Omron CX-Programmer project NewProject (CX-Programmer 9.61)

# PLC AX10: CP1H XA

## Global symbols (name address type ; comment)
0.00 BOOL  ; SENS_1
0.01 BOOL  ; DETECT
0.02 BOOL  ; SENS_2
0.03 BOOL  ; Z_MOV
0.04 BOOL  ; X_MOV
0.05 BOOL  ; START_BT
100.00 BOOL  ; CON
100.01 BOOL  ; Z_AXIS
100.02 BOOL  ; GRAB
100.03 BOOL  ; X_AXIS
100.04 BOOL  ; ROLL
100.05 BOOL  ; CONV_2
100.06 BOOL  ; CONV_3
10.00 BOOL  ; O1
10.01 BOOL  ; O2
10.02 BOOL  ; O3
10.03 BOOL  ; O4
10.04 BOOL  ; O5
T0000 BOOL  ; TIM_1
T0001 BOOL  ; TIM_2
T0002 BOOL  ; TIM_3
T0003 BOOL  ; TIM_4
T0004 BOOL  ; TIM_5
T0005 BOOL  ; TIM_6
T0006 BOOL  ; TIM_7
T0008 BOOL  ; TIM_8
T0009 BOOL  ; TIM_9

## Program NewProgram1 (cyclic task 0)
Local symbols
TOO6 BOOL

### Section Section1

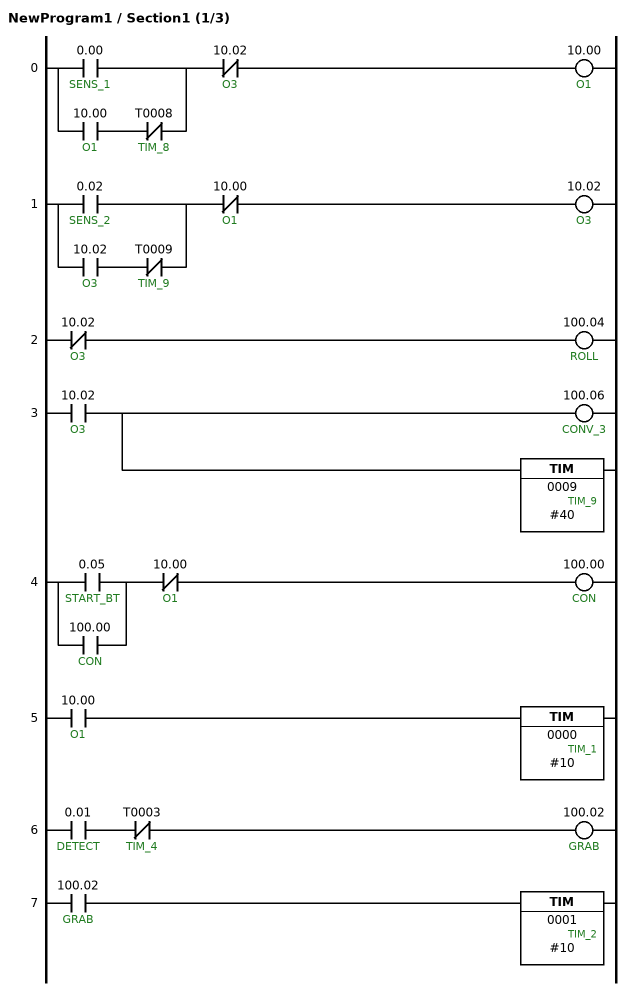
; rung 0
LD 0.00  ; SENS_1
LD 10.00  ; O1
ANDNOT T0008  ; TIM_8
ORLD
ANDNOT 10.02  ; O3
OUT 10.00  ; O1
; rung 1
LD 0.02  ; SENS_2
LD 10.02  ; O3
ANDNOT T0009  ; TIM_9
ORLD
ANDNOT 10.00  ; O1
OUT 10.02  ; O3
; rung 2
LDNOT 10.02  ; O3
OUT 100.04  ; ROLL
; rung 3
LD 10.02  ; O3
OUT 100.06  ; CONV_3
TIM 0009 #40  ; TIM_9
; rung 4
LD 0.05  ; START_BT
OR 100.00  ; CON
ANDNOT 10.00  ; O1
OUT 100.00  ; CON
; rung 5
LD 10.00  ; O1
TIM 0000 #10  ; TIM_1
; rung 6
LD 0.01  ; DETECT
ANDNOT T0003  ; TIM_4
OUT 100.02  ; GRAB
; rung 7
LD 100.02  ; GRAB
TIM 0001 #10  ; TIM_2

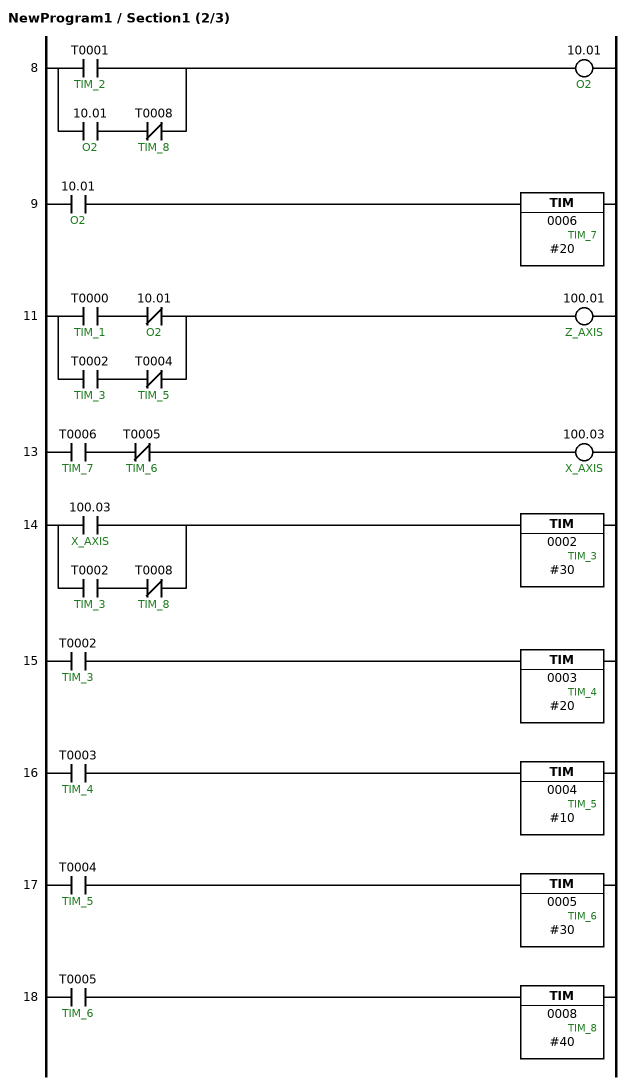
; rung 8
LD T0001  ; TIM_2
LD 10.01  ; O2
ANDNOT T0008  ; TIM_8
ORLD
OUT 10.01  ; O2
; rung 9
LD 10.01  ; O2
TIM 0006 #20  ; TIM_7
; rung 11
LD T0000  ; TIM_1
ANDNOT 10.01  ; O2
LD T0002  ; TIM_3
ANDNOT T0004  ; TIM_5
ORLD
OUT 100.01  ; Z_AXIS
; rung 13
LD T0006  ; TIM_7
ANDNOT T0005  ; TIM_6
OUT 100.03  ; X_AXIS
; rung 14
LD 100.03  ; X_AXIS
LD T0002  ; TIM_3
ANDNOT T0008  ; TIM_8
ORLD
TIM 0002 #30  ; TIM_3
; rung 15
LD T0002  ; TIM_3
TIM 0003 #20  ; TIM_4
; rung 16
LD T0003  ; TIM_4
TIM 0004 #10  ; TIM_5
; rung 17
LD T0004  ; TIM_5
TIM 0005 #30  ; TIM_6
; rung 18
LD T0005  ; TIM_6
TIM 0008 #40  ; TIM_8

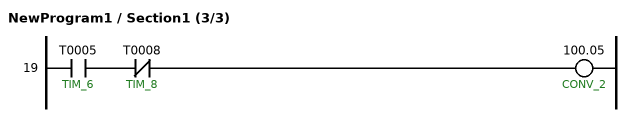
; rung 19
LD T0005  ; TIM_6
ANDNOT T0008  ; TIM_8
OUT 100.05  ; CONV_2

### Section END
; rung 0
END(001)